# EPICS substitutions: lsredis/iocBoot/iocvxWorks/canberra_13.substitutions
file "$(MCA)/mcaApp/Db/simple_mca.db"
{
pattern
{P           M       DTYP           INP         PREC  CHANS}
{lsredis:med:   mca1  "asynMCA"   "@asyn(AIM2/1 0)"    3  2048}
{lsredis:med:   mca2  "asynMCA"   "@asyn(AIM2/1 1)"    3  2048}
{lsredis:med:   mca3  "asynMCA"   "@asyn(AIM2/1 2)"    3  2048}
{lsredis:med:   mca4  "asynMCA"   "@asyn(AIM2/2 0)"    3  2048}
{lsredis:med:   mca5  "asynMCA"   "@asyn(AIM2/2 1)"    3  2048}
{lsredis:med:   mca6  "asynMCA"   "@asyn(AIM2/2 2)"    3  2048}
{lsredis:med:   mca7  "asynMCA"   "@asyn(AIM3/1 0)"    3  2048}
{lsredis:med:   mca8  "asynMCA"   "@asyn(AIM3/1 1)"    3  2048}
{lsredis:med:   mca9  "asynMCA"   "@asyn(AIM3/1 2)"    3  2048}
{lsredis:med:   mca10 "asynMCA"   "@asyn(AIM3/2 0)"    3  2048}
{lsredis:med:   mca11 "asynMCA"   "@asyn(AIM3/3 1)"    3  2048}
{lsredis:med:   mca12 "asynMCA"   "@asyn(AIM3/4 2)"    3  2048}
{lsredis:med:   mca13 "asynMCA"   "@asyn(AIM3/2 3)"    3  2048}
{lsredis:med:   mca0  "Soft Channel"   ""     3  2048}
}

file "$(MCA)/mcaApp/Db/icb_amp.db"
{
pattern
{P			AMP		PORT}
{lsredis:med:	amp1	"icbAmp1"}
{lsredis:med:	amp2	"icbAmp2"}
{lsredis:med:	amp3	"icbAmp3"}
{lsredis:med:	amp4	"icbAmp4"}
{lsredis:med:	amp5	"icbAmp5"}
{lsredis:med:	amp6	"icbAmp6"}
{lsredis:med:	amp7	"icbAmp7"}
{lsredis:med:	amp8	"icbAmp8"}
{lsredis:med:	amp9	"icbAmp9"}
{lsredis:med:	amp10	"icbAmp10"}
{lsredis:med:	amp11	"icbAmp11"}
{lsredis:med:	amp12	"icbAmp12"}
{lsredis:med:	amp13	"icbAmp13"}
}

file "$(MCA)/mcaApp/Db/icb_adc.db"
{
pattern
{P			ADC		PORT}
{lsredis:med:	adc1	"icbAdc1"}
{lsredis:med:	adc2	"icbAdc2"}
{lsredis:med:	adc3	"icbAdc3"}
{lsredis:med:	adc4	"icbAdc4"}
}

file "$(MCA)/mcaApp/Db/icb_hvps.db"
{
pattern
{P			HVPS	LIMIT	PORT}
{lsredis:med:	hvps1	1000	"icbHvps1"}
}
